// TIA Portal V17 export
// export: Created 2025-03-05T08:01:01.5855261Z, ExportSetting WithDefaults, DisplayName Totally Integrated Automation Portal, DisplayVersion V17 Update 8, DisplayName TIA Portal Openness, DisplayVersion V17 Update 8, DisplayName TIA Portal Version Control Interface, DisplayVersion V17, DisplayName SINAMICS Startdrive Advanced, DisplayVersion V17 SP2, DisplayName SINAMICS Startdrive G110M, G120, G120C, G120D, G120P, G115D, DisplayVersion V17 SP2, DisplayName SINAMICS Startdrive G130, G150, S120, S150, SINAMICS MV, S210, DisplayVersion V17 SP2, DisplayName STEP 7 Professional, DisplayVersion V17 Update 8, DisplayName SINUMERIK ONE STEP 7 Toolbox, DisplayVersion V17 Update 12, DisplayName SINUMERIK 840D sl STEP 7 Toolbox, DisplayVersion V17 Update 12, DisplayName STEP 7 Safety, DisplayVersion V17 Update 6, DisplayName WinCC Advanced, DisplayVersion V17 Update 8
DATA_BLOCK "LTLP_NcHMIProInterfaceData"   // DB549
{ S7_Optimized_Access := 'FALSE'; DB_Accessible_From_OPC_UA := 'FALSE' }
VERSION : 0.1
// stored: AutoNumber true, DBAccessibleFromOPCUA false, DBAccessibleFromWebserver true, InstanceOfName LTLP_typeNcHmiProInterface, InstanceOfType UDT, IsOnlyStoredInLoadMemory false, IsWriteProtectedInAS false
"LTLP_typeNcHmiProInterface"
   // VAR RETAIN
   //    reserved0 : Array[0..3] of Byte;
   //    bagDataSpecification { S7_SetPoint := 'True'} : "LTLP_typeModeGroupDataToNC";
   //    bagDataFeedback { S7_SetPoint := 'True'} : "LTLP_typeModeGroupDataFromNC";
   //    channelDataSpecification { S7_SetPoint := 'True'} : "LTLP_typeChannelDataToNC";
   //    channelDataFeedback { S7_SetPoint := 'True'} : "LTLP_typeChannelDataFromNC";
   //    axisSpecification { S7_SetPoint := 'True'} : "LTLP_typeAxisDataToNC";
   //    axisFeedback { S7_SetPoint := 'True'} : "LTLP_typeAxisDataFromNC";
   //    fromHMI1 : Struct
   //       axisPosition : Array[1..17] of Char;
   //       hmiSync : Byte;
   //       reserved19 : Array[19..28] of Byte;
   //    END_STRUCT;
   //    versionAxisScreen : Word;
   //    versionPlcBlock : Word;
   //    reserved52_0 : Array[52..57] of Byte;
   //    fromHMI : Struct
   //       axisSelectionActiv : Bool;
   //       transformationActiv : Bool;
   //       axisIsGeoAxis : Bool;
   //       reserve0p3 : Bool;
   //       reserve0p4 : Bool;
   //       reserve0p5 : Bool;
   //       transmitActiv : Bool;
   //       reserve0p7 : Bool;
   //       hmiSync : Byte;
   //       axisNoNc : Byte;
   //       axisNoMcp : Byte;
   //       ht8UserKeys : Word;
   //       axisName : Array[1..17] of Char;
   //    END_STRUCT;
   //    fromPlc : Struct
   //       axisSelectionScreen : Byte;
   //       plcSync : Byte;
   //       axisNoMcp : Byte;
   //       bag : Byte;
   //       channelNo : Byte;
   //       activateHeaderDisplay : Bool;
   //       axisTakeoverDisabled : Bool;
   //       incrementVarableActive : Bool;
   //       mppDAGNotAvailable : Bool;
   //       mppNotAvailable : Bool;
   //       mcpNotAvailable : Bool;
   //       ht8NotAvailable : Bool;
   //       ht2NotAvailable : Bool;
   //       ht8UserKeys : Word;
   //       ht2IsActiv : Bool;
   //       reserved81 : Bool;
   //       reserved82 : Bool;
   //       reserved83 : Bool;
   //       reserved84 : Bool;
   //       reserved85 : Bool;
   //       reserved86 : Bool;
   //       reserved87 : Bool;
   //       reserved9 : Array[9..15] of Byte;
   //    END_STRUCT;
   //    internalStorageData : Struct
   //       localStat : Struct
   //          spSingleblockChannel : Bool;
   //          impulsKeySingleblock : Bool;
   //          negTriggerKeySingleblock : Bool;
   //          posTriggerTLfunctionSingleStep : Bool;
   //          negTriggerTLfunctionSingleStep : Bool;
   //          posTriggerAxisSwitch : Bool;
   //          operationModeIncrementVariable : Bool;
   //          initReady : Bool;
   //          posTriggerNCModeManual : Bool;
   //          staticNCModeManual : Bool;
   //          mcsWcsOld : Bool;
   //          posTriggerTransformation : Bool;
   //          reserve_2p3 : Bool;
   //          reserve_2p4 : Bool;
   //          reserve_2p5 : Bool;
   //          reserve_2p6 : Bool;
   //          reserve_2p7 : Bool;
   //          operationModeOld : Byte;
   //          posTriggerAxisNext : Bool;
   //          impulsAxisNext : Bool;
   //          axisNextActive : Bool;
   //          reserveNextPlus : Bool;
   //          posTriggerAxisPrevious : Bool;
   //          impulseAxisPrevious : Bool;
   //          axisPreviousActive : Bool;
   //          reserveAxisPrevious : Bool;
   //       END_STRUCT;
   //       axis : Byte;
   //       axisret : Byte;
   //       channel : Byte;
   //       channelRet : Byte;
   //       bag : Byte;
   //       bagRet : Byte;
   //       hmiSyncRet : Byte;
   //       axisPlusMinus1 : Byte;
   //       axisPlusMinus2 : Byte;
   //    END_STRUCT;
   // END_VAR
BEGIN
END_DATA_BLOCK
